# EPICS substitutions: iocBoot/ioczzz/zedLOreg4.substitutions
file "$(TOP)/zzzApp/Db/zedLOreg.template"
{
pattern
{P,R,C,N, SCAN}
{zzz:,reg4_,4,0,8}
{zzz:,reg4_,4,1,8}
{zzz:,reg4_,4,2,8}
{zzz:,reg4_,4,3,8}
{zzz:,reg4_,4,4,8}
}
